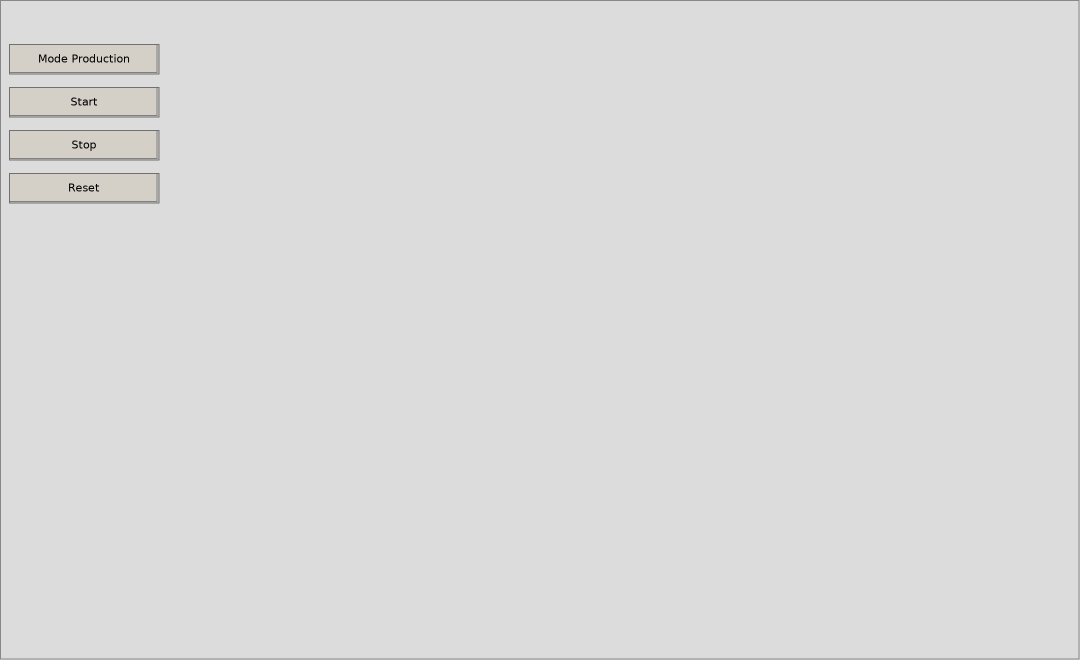
VISUALIZATION Page_Main  // 1080x660
    Button (9,44 150x30), "Mode Production"
        OnMouseClick: execute { GVL_Modules.g_fbHmiMachCtrlsManager.q_eReqMode := E_PackML_Mode.Production; }
    Button (9,87 150x30), "Start", colour toggle: GVL_Modules.g_fbMachCtrlsManager.s_fbDiBtnStart[1].I_bIn
        OnMouseDown: execute { GVL_Modules.g_fbMachCtrlsManager.s_fbDiBtnStart[1].I_bIn := TRUE; }
        OnMouseUp: execute { GVL_Modules.g_fbMachCtrlsManager.s_fbDiBtnStart[1].I_bIn := FALSE; }
    Button (9,130 150x30), "Stop", colour toggle: GVL_Modules.g_fbMachCtrlsManager.s_fbDiBtnStop[1].I_bIn
        OnMouseDown: execute { GVL_Modules.g_fbMachCtrlsManager.s_fbDiBtnStop[1].I_bIn := TRUE; }
        OnMouseUp: execute { GVL_Modules.g_fbMachCtrlsManager.s_fbDiBtnStop[1].I_bIn := FALSE; }
    Button (9,173 150x30), "Reset", colour toggle: GVL_Modules.g_fbAlarmManager.s_bCmdResetFromDebug
        OnMouseDown: execute { GVL_Modules.g_fbAlarmManager.s_bCmdResetFromDebug := TRUE; }
        OnMouseUp: execute { GVL_Modules.g_fbAlarmManager.s_bCmdResetFromDebug := FALSE; }
END_VISUALIZATION

(* stored: Version 1.1.0.1, ProductVersion 3.1.4026.13
   Visu Page_Main: Id {d6edb6b5-3389-4935-ba25-f59ab80f47dd} *)
